// TwinCAT 3 PLC project HARTL_PowerLink_v2_01
// ProgramVersion: 3.1.4023.0
// libraries:
//   EfficientIO Communicator, * (EfficientIO)
//   EfficientIO ModbusTCP, * (EfficientIO)
//   Lynus Energy Basic, * (Lynus AG)
//   Lynus Standards, * (Lynus AG)
//   Tc2_BABasic, * (Beckhoff Automation GmbH)
//   Tc2_ModbusSrv, * (Beckhoff Automation GmbH)
//   Tc2_Standard, * (Beckhoff Automation GmbH)
//   Tc2_System, * (Beckhoff Automation GmbH)
//   Tc2_Utilities, * (Beckhoff Automation GmbH)
//   Tc3_Module, * (Beckhoff Automation GmbH)
// project tree:
//   / FastTask.TcTTO (not stored), MiddleTask.TcTTO, SlowTask.TcTTO
//   FBs/ FB_EM24_DIN.TcPOU, FB_Enphase.TcPOU (not stored), FB_Enphase_Helper.TcPOU, FB_ModBus_2Registers.TcPOU
//   POUs/ prgBattery.TcPOU, prgCalc.TcPOU, prgComEffIO.TcPOU, prgEM.TcPOU, prgEMS.TcPOU, prgEnphase.TcPOU (not stored), prgPV.TcPOU, prgCS.TcPOU, prgRWEffIO.TcPOU (not stored), prgSystemTime.TcPOU, prgVarEffIO.TcPOU (not stored)
// real-time tasks:
//   TASK MiddleTask: cycle T#10ms, priority 20, ADS port 350
//   TASK FastTask: cycle T#5ms, priority 19, ADS port 351
//   TASK SlowTask: cycle T#20ms, priority 21, ADS port 352
// I/O:
//   DEVICE Device 1 (Beckhoff CCAT)
//   DEVICE Device 2 (CX-BK)
//     Box 1 (CX-BK)
// variable links:
//   HARTL_PowerLink_v2_01/HARTL_PowerLink_v2_01 Instance <-> Device 2 (CX-BK)/Box 1 (CX-BK)
//     MiddleTask Inputs/prgEM.fbEM1.fbKL3403.byStateCH1 <-> Term 2 (KL3403)/Channel 1/State
//     MiddleTask Inputs/prgEM.fbEM1.fbKL3403.byStateCH2 <-> Term 2 (KL3403)/Channel 2/State
//     MiddleTask Inputs/prgEM.fbEM1.fbKL3403.byStateCH3 <-> Term 2 (KL3403)/Channel 3/State
//     MiddleTask Inputs/prgEM.fbEM2.fbKL3403.byStateCH1 <-> Term 3 (KL3403)/Channel 1/State
//     MiddleTask Inputs/prgEM.fbEM2.fbKL3403.byStateCH2 <-> Term 3 (KL3403)/Channel 2/State
//     MiddleTask Inputs/prgEM.fbEM2.fbKL3403.byStateCH3 <-> Term 3 (KL3403)/Channel 3/State
//     MiddleTask Inputs/prgEM.fbEM3.fbKL3403.byStateCH1 <-> Term 4 (KL3403)/Channel 1/State
//     MiddleTask Inputs/prgEM.fbEM3.fbKL3403.byStateCH2 <-> Term 4 (KL3403)/Channel 2/State
//     MiddleTask Inputs/prgEM.fbEM3.fbKL3403.byStateCH3 <-> Term 4 (KL3403)/Channel 3/State
//     MiddleTask Inputs/prgEM.fbEM4.fbKL3403.byStateCH1 <-> Term 5 (KL3403)/Channel 1/State
//     MiddleTask Inputs/prgEM.fbEM4.fbKL3403.byStateCH2 <-> Term 5 (KL3403)/Channel 2/State
//     MiddleTask Inputs/prgEM.fbEM4.fbKL3403.byStateCH3 <-> Term 5 (KL3403)/Channel 3/State
//     MiddleTask Inputs/prgEM.fbEM1.fbKL3403.iDataInCH1 <-> Term 2 (KL3403)/Channel 1/Data In
//     MiddleTask Inputs/prgEM.fbEM1.fbKL3403.iDataInCH2 <-> Term 2 (KL3403)/Channel 2/Data In
//     MiddleTask Inputs/prgEM.fbEM1.fbKL3403.iDataInCH3 <-> Term 2 (KL3403)/Channel 3/Data In
//     MiddleTask Inputs/prgEM.fbEM2.fbKL3403.iDataInCH1 <-> Term 3 (KL3403)/Channel 1/Data In
//     MiddleTask Inputs/prgEM.fbEM2.fbKL3403.iDataInCH2 <-> Term 3 (KL3403)/Channel 2/Data In
//     MiddleTask Inputs/prgEM.fbEM2.fbKL3403.iDataInCH3 <-> Term 3 (KL3403)/Channel 3/Data In
//     MiddleTask Inputs/prgEM.fbEM3.fbKL3403.iDataInCH1 <-> Term 4 (KL3403)/Channel 1/Data In
//     MiddleTask Inputs/prgEM.fbEM3.fbKL3403.iDataInCH2 <-> Term 4 (KL3403)/Channel 2/Data In
//     MiddleTask Inputs/prgEM.fbEM3.fbKL3403.iDataInCH3 <-> Term 4 (KL3403)/Channel 3/Data In
//     MiddleTask Inputs/prgEM.fbEM4.fbKL3403.iDataInCH1 <-> Term 5 (KL3403)/Channel 1/Data In
//     MiddleTask Inputs/prgEM.fbEM4.fbKL3403.iDataInCH2 <-> Term 5 (KL3403)/Channel 2/Data In
//     MiddleTask Inputs/prgEM.fbEM4.fbKL3403.iDataInCH3 <-> Term 5 (KL3403)/Channel 3/Data In
//     MiddleTask Inputs/prgEM.fbKBusState.uiKBusState_OUT <-> Inputs/State
//     MiddleTask Outputs/prgEM.fbEM1.fbKL3403.byCntrCH1 <-> Term 2 (KL3403)/Channel 1/Ctrl
//     MiddleTask Outputs/prgEM.fbEM1.fbKL3403.byCntrCH2 <-> Term 2 (KL3403)/Channel 2/Ctrl
//     MiddleTask Outputs/prgEM.fbEM1.fbKL3403.byCntrCH3 <-> Term 2 (KL3403)/Channel 3/Ctrl
//     MiddleTask Outputs/prgEM.fbEM2.fbKL3403.byCntrCH1 <-> Term 3 (KL3403)/Channel 1/Ctrl
//     MiddleTask Outputs/prgEM.fbEM2.fbKL3403.byCntrCH2 <-> Term 3 (KL3403)/Channel 2/Ctrl
//     MiddleTask Outputs/prgEM.fbEM2.fbKL3403.byCntrCH3 <-> Term 3 (KL3403)/Channel 3/Ctrl
//     MiddleTask Outputs/prgEM.fbEM3.fbKL3403.byCntrCH1 <-> Term 4 (KL3403)/Channel 1/Ctrl
//     MiddleTask Outputs/prgEM.fbEM3.fbKL3403.byCntrCH2 <-> Term 4 (KL3403)/Channel 2/Ctrl
//     MiddleTask Outputs/prgEM.fbEM3.fbKL3403.byCntrCH3 <-> Term 4 (KL3403)/Channel 3/Ctrl
//     MiddleTask Outputs/prgEM.fbEM4.fbKL3403.byCntrCH1 <-> Term 5 (KL3403)/Channel 1/Ctrl
//     MiddleTask Outputs/prgEM.fbEM4.fbKL3403.byCntrCH2 <-> Term 5 (KL3403)/Channel 2/Ctrl
//     MiddleTask Outputs/prgEM.fbEM4.fbKL3403.byCntrCH3 <-> Term 5 (KL3403)/Channel 3/Ctrl
//     MiddleTask Outputs/prgEMS.bQ1State <-> Term 6 (KL2012)/Channel 1/Output
//     MiddleTask Outputs/prgEMS.bQ2State <-> Term 6 (KL2012)/Channel 2/Output
//     MiddleTask Outputs/prgEMS.bQ3State <-> Term 7 (KL2012)/Channel 1/Output
//     MiddleTask Outputs/prgEMS.bQ4State <-> Term 7 (KL2012)/Channel 2/Output

CONFIGURATION HARTL_PowerLink_v2_01
    RESOURCE PLC ON TwinCAT3
        TASK MiddleTask(INTERVAL := T#10ms, PRIORITY := 20);
        TASK SlowTask(INTERVAL := T#20ms, PRIORITY := 21);
        PROGRAM prgEM WITH MiddleTask : prgEM;
        PROGRAM prgEMS WITH MiddleTask : prgEMS;
        PROGRAM prgSystemTime WITH MiddleTask : prgSystemTime;
        PROGRAM prgCS WITH MiddleTask : prgCS;
        PROGRAM prgCalc WITH MiddleTask : prgCalc;
        PROGRAM prgComEffIO WITH SlowTask : prgComEffIO;
    END_RESOURCE
END_CONFIGURATION

// ---- POUs/prgEM.TcPOU
PROGRAM prgEM
VAR
	fbKBusState		: FB_K_Bus_State;
	fbEM1			: FB_EM_Beckhoff_KL3403;
	fbEM1Counter	: FB_EnergyCounter;
	fbEM2			: FB_EM_Beckhoff_KL3403;
	fbEM2Counter	: FB_EnergyCounter;
	fbEM3			: FB_EM_Beckhoff_KL3403;
	fbEM3Counter	: FB_EnergyCounter;
	fbEM4			: FB_EM_Beckhoff_KL3403;
	fbEM4Counter	: FB_EnergyCounter;
	lrPowerEM1		: LREAL;						//{#lynus.ag#()}
	lrPowerEM2		: LREAL;						//{#lynus.ag#()}
	lrPowerEM3		: LREAL;						//{#lynus.ag#()}
	lrPowerEM4		: LREAL;						//{#lynus.ag#()}
	lr_InputVoltage_L1N		: LREAL;						//{#lynus.ag#()}
	lr_InputVoltage_L2N		: LREAL;						//{#lynus.ag#()}
	lr_InputVoltage_L3N		: LREAL;						//{#lynus.ag#()}
	lr_InputVoltage_L1L2	: LREAL;						//{#lynus.ag#()}
	lr_InputVoltage_L2L3	: LREAL;						//{#lynus.ag#()}
	lr_InputVoltage_L3L1	: LREAL;						//{#lynus.ag#()}


END_VAR
VAR PERSISTENT
	lrCounterEM1	: LREAL;						//{#lynus.ag#()}
	lrCounterEM2	: LREAL;						//{#lynus.ag#()}
	lrCounterEM3	: LREAL;						//{#lynus.ag#()}
	lrCounterEM4	: LREAL;						//{#lynus.ag#()}
END_VAR

fbKBusState(uiKBusState_OUT=> );

// Base Connection

fbEM1(
	bEnable:= TRUE, 
	bChannel1Invers:= FALSE,
	bChannel2Invers:= FALSE,
	bChannel3Invers:= FALSE,
	uiCurrentTransformerRatioL1:= 64, 
	uiCurrentTransformerRatioL2:= 64, 
	uiCurrentTransformerRatioL3:= 64, 
	uiKBusState_IN:= fbKBusState.uiKBusState_OUT, 
	stDataEMPower=> , 
	stDataEMCounter=> , 
	stDataEMPowerRealTime=> , 
	stDataEMCounterRealTime=> , 
	diNrOfEM_OUT=> );

lrPowerEM1 := fbEM1.stDataEMPower.lrPowerTotal;	
lr_InputVoltage_L1N := fbEM1.stDataEMPower.lrVoltageL1N;
lr_InputVoltage_L2N := fbEM1.stDataEMPower.lrVoltageL2N;
lr_InputVoltage_L3N := fbEM1.stDataEMPower.lrVoltageL3N;
lr_InputVoltage_L1L2 := fbEM1.stDataEMPower.lrVoltageL1L2;
lr_InputVoltage_L2L3 := fbEM1.stDataEMPower.lrVoltageL2L3;
lr_InputVoltage_L3L1 := fbEM1.stDataEMPower.lrVoltageL3L1;

fbEM1Counter(
	byActiveTariff:= 1, 
	lrPowerInput:= lrPowerEM1, 
	lrTotalCounterEnergy_Consumption=> , 
	lrTotalCounterEnergy_Production=> , 
	lrCounterEnergyT1_Consumption=> , 
	lrCounterEnergyT2_Consumption=> , 
	lrCounterEnergyT1_Production=> , 
	lrCounterEnergyT2_Production=> );
	
IF fbEM1Counter.lrTotalCounterEnergy_Consumption > lrCounterEM1 THEN  	
	lrCounterEM1 := fbEM1Counter.lrTotalCounterEnergy_Consumption;
END_IF

// Output1, 3x400V 32A, CEE32

fbEM2(
	bEnable:= TRUE, 
	bChannel1Invers:= FALSE,
	bChannel2Invers:= FALSE,
	bChannel3Invers:= FALSE,
	uiCurrentTransformerRatioL1:= 35, 
	uiCurrentTransformerRatioL2:= 35, 
	uiCurrentTransformerRatioL3:= 35, 
	uiKBusState_IN:= fbKBusState.uiKBusState_OUT, 
	stDataEMPower=> , 
	stDataEMCounter=> , 
	stDataEMPowerRealTime=> , 
	stDataEMCounterRealTime=> , 
	diNrOfEM_OUT=> );

lrPowerEM2 := fbEM2.stDataEMPower.lrPowerTotal;	

fbEM2Counter(
	byActiveTariff:= 1, 
	lrPowerInput:= lrPowerEM2, 
	lrTotalCounterEnergy_Consumption=> , 
	lrTotalCounterEnergy_Production=> , 
	lrCounterEnergyT1_Consumption=> , 
	lrCounterEnergyT2_Consumption=> , 
	lrCounterEnergyT1_Production=> , 
	lrCounterEnergyT2_Production=> );
	
IF fbEM2Counter.lrTotalCounterEnergy_Consumption > lrCounterEM2 THEN  	
	lrCounterEM2 := fbEM2Counter.lrTotalCounterEnergy_Consumption;
END_IF


// Output2, 3x400V 32A, CEE32

fbEM3(
	bEnable:= TRUE, 
	bChannel1Invers:= FALSE,
	bChannel2Invers:= FALSE,
	bChannel3Invers:= FALSE,
	uiCurrentTransformerRatioL1:= 35, 
	uiCurrentTransformerRatioL2:= 35, 
	uiCurrentTransformerRatioL3:= 35, 
	uiKBusState_IN:= fbKBusState.uiKBusState_OUT, 
	stDataEMPower=> , 
	stDataEMCounter=> , 
	stDataEMPowerRealTime=> , 
	stDataEMCounterRealTime=> , 
	diNrOfEM_OUT=> );

lrPowerEM3 := fbEM3.stDataEMPower.lrPowerTotal;	

fbEM3Counter(
	byActiveTariff:= 1, 
	lrPowerInput:= lrPowerEM3, 
	lrTotalCounterEnergy_Consumption=> , 
	lrTotalCounterEnergy_Production=> , 
	lrCounterEnergyT1_Consumption=> , 
	lrCounterEnergyT2_Consumption=> , 
	lrCounterEnergyT1_Production=> , 
	lrCounterEnergyT2_Production=> );
	
IF fbEM3Counter.lrTotalCounterEnergy_Consumption > lrCounterEM3 THEN  	
	lrCounterEM3 := fbEM3Counter.lrTotalCounterEnergy_Consumption;
END_IF


// Output3, 3x400V 16A, CEE16

fbEM4(
	bEnable:= TRUE, 
	bChannel1Invers:= FALSE,
	bChannel2Invers:= FALSE,
	bChannel3Invers:= FALSE,
	uiCurrentTransformerRatioL1:= 35, 
	uiCurrentTransformerRatioL2:= 35, 
	uiCurrentTransformerRatioL3:= 35, 
	uiKBusState_IN:= fbKBusState.uiKBusState_OUT, 
	stDataEMPower=> , 
	stDataEMCounter=> , 
	stDataEMPowerRealTime=> , 
	stDataEMCounterRealTime=> , 
	diNrOfEM_OUT=> );

lrPowerEM4 := fbEM4.stDataEMPower.lrPowerTotal;	

fbEM4Counter(
	byActiveTariff:= 1, 
	lrPowerInput:= lrPowerEM4, 
	lrTotalCounterEnergy_Consumption=> , 
	lrTotalCounterEnergy_Production=> , 
	lrCounterEnergyT1_Consumption=> , 
	lrCounterEnergyT2_Consumption=> , 
	lrCounterEnergyT1_Production=> , 
	lrCounterEnergyT2_Production=> );
	
IF fbEM4Counter.lrTotalCounterEnergy_Consumption > lrCounterEM4 THEN  	
	lrCounterEM4 := fbEM4Counter.lrTotalCounterEnergy_Consumption;
END_IF

END_PROGRAM

// ---- POUs/prgEMS.TcPOU
PROGRAM prgEMS
VAR
	// Q1, 3x400V 32A, CEE32
	fbQ1						: FB_Light;
	bQ1On						: BOOL;						//{#lynus.ag#()}
	bQ1Off						: BOOL;						//{#lynus.ag#()}
	bQ1State	AT%Q*			: BOOL;						//{#lynus.ag#()}
	// Q2, 3x400V 32A, CEE32
	fbQ2						: FB_Light;
	bQ2On						: BOOL;						//{#lynus.ag#()}
	bQ2Off						: BOOL;						//{#lynus.ag#()}
	bQ2State	AT%Q*			: BOOL;						//{#lynus.ag#()}
	// Q3, 3x400V 16A, CEE16
	fbQ3						: FB_Light;	
	bQ3On						: BOOL;						//{#lynus.ag#()}
	bQ3Off						: BOOL;						//{#lynus.ag#()}
	bQ3State	AT%Q*			: BOOL;						//{#lynus.ag#()}
	// Q4, 3x400V 16A, CEE16, EV Charging
	fbQ4						: FB_Light;
	bQ4On						: BOOL;						//{#lynus.ag#()}
	bQ4Off						: BOOL;						//{#lynus.ag#()}
	bQ4State	AT%Q*			: BOOL;						//{#lynus.ag#()}
	
	// Automatic PV-Inverter Shutdown
	fbNFS_PV					: FB_WeeklyTimeSwitch;
	fbCalcSunriseSunset   		: FB_CalcSunriseSunset;
	todSunrise            		: TOD;
	todSunset             		: TOD;
END_VAR
VAR PERSISTENT
	bEnableNFS_PV				: BOOL;						//{#lynus.ag#()}
END_VAR

// To-Do:
// adopt Longitude and Latitude
// set bEdgeOn and bEdgeOff to correct Q Variables


// Output Controls
fbQ1(bOn:=bQ1On, bOff:=bQ1Off, bLight=>bQ1State);
fbQ2(bOn:=bQ2On, bOff:=bQ2Off, bLight=>bQ2State);
fbQ3(bOn:=bQ3On, bOff:=bQ3Off, bLight=>bQ3State);
fbQ4(bOn:=bQ4On, bOff:=bQ4Off, bLight=>bQ4State);

// Sunrise, Sunset calc
IF prgSystemTime.bSystemTimeValid THEN

	fbCalcSunriseSunset(
		fDegreeOfLongitude := 11.5820,   (* Longitude of Munich, Lochhausen *)
        fDegreeOfLatitude := 48.1351,   (* Latitude of Munich, Lochhausen *)
    	fReferenceMeridian := 15.0,  (* Central European Time *)
        dCurrentDate := DT_TO_DATE(prgSystemTime.dtSystemTime),
        todSunrise => todSunrise,
        todSunset => todSunset);
END_IF

// Automatic PV-Inverter Shutdown
IF prgSystemTime.bSystemTimeValid THEN
	fbNFS_PV(
		bEnable:=bEnableNFS_PV, 
		tCurrentDateTime:=prgSystemTime.dtSystemTime, 
		tSwitchOnTime:=todSunrise, 
		tSwitchOffTime:=todSunset, 
		bSunday:=TRUE, 
		bMonday:=TRUE, 
		bTuesday:=TRUE, 
		bWednesday:=TRUE, 
		bThursday:=TRUE, 
		bFriday:=TRUE, 
		bSaturday:=TRUE,
		bEdgeOn=> ,
		bEdgeOff=> );
END_IF

END_PROGRAM

// ---- POUs/prgSystemTime.TcPOU
PROGRAM prgSystemTime
VAR
	fbGetTime			: NT_GetTime;
	dtSystemTime		: DT;
	stDateTime			: TIMESTRUCT;
	tonGetTime			: TON;
	nStep				: INT;
	bSystemTimeValid	: BOOL := FALSE;
END_VAR

CASE nStep OF
0:
	tonGetTime(IN:=TRUE, PT:=T#500MS);
	IF (tonGetTime.Q) THEN
		tonGetTime(IN := FALSE);
		nStep:=10;
	END_IF

10:
	fbGetTime(NETID:='', START:=TRUE, TMOUT:=T#2S);
	IF (NOT fbGetTime.BUSY) THEN
		stDateTime := fbGetTime.TIMESTR;
		dtSystemTime := SYSTEMtimE_TO_DT(fbGetTime.TIMESTR);
		fbGetTime(START := FALSE);
		bSystemTimeValid := TRUE;
		nStep := 0;
	END_IF	
END_CASE

END_PROGRAM

// ---- POUs/prgCS.TcPOU
PROGRAM prgCS
VAR
	fbCS						: FB_EM24_DIN;
	fbCSCounter					: FB_EnergyCounter;
	lrPowerCS					: LREAL;						//{#lynus.ag#()}
	// udintErrorWarningCS			: UDINT;
END_VAR
VAR PERSISTENT
	lrCounterCS					: LREAL;						//{#lynus.ag#()}
	lrCounterCSeIO				: LREAL;						//{#lynus.ag#()}
END_VAR

// To-Do:
// adopt FB Declaration, change to new FB for ENERGYMID
// adopt FB Definition, change to correct in/out Vars for ENERGYMID
// correct lrPowerCS definition
// correct lrCounterCS definition
// correct byErrorWarningCS definition

fbCS(
	m_Enable:= TRUE, 
	str_IPAdress:= '192.168.1.20',  
	real_RealPower_kW=> lrPowerCS, 
	real_RealPowerL1_kW=> , 
	real_RealPowerL2_kW=> , 
	real_RealPowerL3_kW=> , 
	real_ReactivePower_kVAr=> , 
	real_ApparentPower_kVA=> , 
	real_Frequency_Hz=> , 
	real_VoltageL1N_V=> , 
	real_VoltageL2N_V=> , 
	real_VoltageL3N_V=> , 
	real_VoltageL1L2_V=> , 
	real_VoltageL2L3_V=> , 
	real_VoltageL3L1_V=> , 
	real_CurrentL1_A=> , 
	real_CurrentL2_A=> , 
	real_CurrentL3_A=> , 
	real_EnergyTotal_Import_kWh=> , 
	real_EnergyTotal_Export_kWh=> , 
	real_EnergyTotal_ExportT1_kWh=> , 
	real_EnergyTotal_ExportT2_kWh=> , 
	real_EnergyTotal_ExportT3_kWh=> , 
	real_EnergyTotal_ExportT4_kWh=> , 
	m_PollSuccessful=> , 
	udint_Error_ID=> );



// uErrorWarningCS := fbCS.udint_Error_ID;

// MID conform Counter, read from Energymeter
IF fbCS.real_EnergyTotal_Import_kWh > lrCounterCS THEN  	
	lrCounterCS := fbCS.real_EnergyTotal_Import_kWh;
END_IF

// internal Counter, for comparing purpose
fbCSCounter(
	byActiveTariff:= 1, 
	lrPowerInput:= lrPowerCS, 
	lrTotalCounterEnergy_Consumption=> , 
	lrTotalCounterEnergy_Production=> , 
	lrCounterEnergyT1_Consumption=> , 
	lrCounterEnergyT2_Consumption=> , 
	lrCounterEnergyT1_Production=> , 
	lrCounterEnergyT2_Production=> );
	
IF fbCSCounter.lrTotalCounterEnergy_Consumption > lrCounterCSeIO THEN  	
	lrCounterCSeIO := fbCSCounter.lrTotalCounterEnergy_Consumption;
END_IF

END_PROGRAM

// ---- FBs/FB_EM24_DIN.TcPOU
FUNCTION_BLOCK FB_EM24_DIN
VAR_INPUT PERSISTENT
	m_Enable					: BOOL;						//Enable the Fuctionblock and his logic
	str_IPAdress				: STRING(15);				//IP Adress of the meter
END_VAR
VAR_OUTPUT
	real_RealPower_kW				: REAL;					// Real power in W
	real_RealPowerL1_kW				: REAL;					// Real power in W
	real_RealPowerL2_kW				: REAL;					// Real power in W
	real_RealPowerL3_kW				: REAL;					// Real power in W
	real_ReactivePower_kVAr			: REAL;					// Reactive power in VAr
	real_ApparentPower_kVA			: REAL;					// Apparent power in VA
	real_Frequency_Hz				: REAL;					// Frequency in Hz
	real_VoltageL1N_V				: REAL;					//  Voltage L1-N in V 
	real_VoltageL2N_V				: REAL;					//  Voltage L2-N in V 
	real_VoltageL3N_V				: REAL;					//  Voltage L3-N in V 
	real_VoltageL1L2_V				: REAL;					//  Voltage L1-L2 in V 
	real_VoltageL2L3_V				: REAL;					//  Voltage L2-L3 in V 
	real_VoltageL3L1_V				: REAL;					//  Voltage L3-L1 in V 
	real_CurrentL1_A				: REAL;					//  Current L1 in A
	real_CurrentL2_A				: REAL;					//  Current L2 in A
	real_CurrentL3_A				: REAL;					//  Current L3 in A
	real_EnergyTotal_Import_kWh		: REAL;					// Energy total in Wh
	real_EnergyTotal_Export_kWh		: REAL;					// Energy total in Wh
	real_EnergyTotal_ExportT1_kWh	: REAL;					// Energy total in Wh
	real_EnergyTotal_ExportT2_kWh	: REAL;					// Energy total in Wh
	real_EnergyTotal_ExportT3_kWh	: REAL;					// Energy total in Wh
	real_EnergyTotal_ExportT4_kWh	: REAL;					// Energy total in Wh
	
	m_PollSuccessful				: BOOL;					// Poll succesfull		
	udint_Error_ID					: UDINT;				// ERR ID FB_MBReadRegs
END_VAR
VAR
	{attribute 'hide'}
	w_Adress					: WORD;						//modbus adress
	{attribute 'hide'}
	usint_Quantity				: USINT;					//Number of Words to get polled, max 100
	{attribute 'hide'}
	fbConvertWordToDword		: FB_CV_WORD_TO_DWORD;			//Convert Word to Dword
	{attribute 'hide'}
	usintSign					: USINT;						// converstion dword to real	
	{attribute 'hide'}
	intExponent					: INT;							// converstion dword to real
	{attribute 'hide'}
	realMantisse				: REAL;							// converstion dword to real
	{attribute 'hide'}
	timer_Delay					: TON;						//Timer for Delay between Requests
	{attribute 'hide'}
	timer_DelayStart			: TON;						//Timer to start the state machine with Delay after enabling or after the system ist restartet
	{attribute 'hide'}
	timer_TimeOut				: TON;						//Timer for Timeout MB Read
	{attribute 'hide'}
	iStateModbusRead			: INT;						//State machine for read out Data over Modbus RTU
	{attribute 'hide'}
	fbMBRead_FC3				: FB_MBReadRegs  ;		//Modbus Read Function (FC3)
	{attribute 'hide'}
	ftrig_PEnable				: f_trig;					//Internal positive Edge
	{attribute 'hide'}
	iStateModbusError			: INT;						//State machine for error out Data over Modbus TCP/IP	
	{attribute 'hide'}
	FPError_FC_3				: R_TRIG;					//Internal positive Edge
	{attribute 'hide'}
	arrBuffer_FC3				: ARRAY[0..10] OF WORD;		//Buffer with Data from FC3
	{attribute 'hide'}
	arrBuffer_Received			: ARRAY[0..120] OF WORD;		//Total received Data
	{attribute 'hide'}
	timer_Connection_ok			: TON;
	{attribute 'hide'}
	int_Data_Received			: INT;
	{attribute 'hide'}
	m_MBTCPError				: BOOL;
	{attribute 'hide'}
	int_Data_Received_old		: INT;
	{attribute 'hide'}
	timer_Connection_ok_TOF	: TOF;
	{attribute 'hide'}
	m_Poll_ok: BOOL;
	{attribute 'hide'}
	timer_Wait: Ton;
	{attribute 'hide'}
	int_TimeoutError: INT;
	{attribute 'hide'}
	int_FC4Error: INT;
	{attribute 'hide'}
	i: INT;
END_VAR

// v0.1 by Stefan Lackner 20230330
// tested, but not with current flowing. Votlages & frequency working.
// reads out Carlo Gavazzi EM24-Din Multimeter


(*--------------------------------------------------------------------------------------------Limits-------------------------------------------------------------------------------------*)
w_Adress := LIMIT(0,w_Adress,65000);
usint_Quantity := LIMIT(1,usint_Quantity,100);
	
(*--------------------------------------------------------------------------------------------State Machine Read--------------------------------------------------------------------------------------*)

//Timer for Delay
timer_Delay(IN:= , PT:= T#50MS, Q=> , ET=> );

//Timeout Timer is dissabled when the Init Step is aktiv or the function is not enabled
IF iStateModbusRead = 0 OR NOT m_Enable THEN 
	timer_Timeout.IN := FALSE; 
END_IF
timer_Timeout(IN:= , PT:= T#1S, Q=> , ET=> );

//Enable with Delay that not all sockets have to be created at the same time
timer_DelayStart(IN:= m_Enable, PT:= T#1S, Q=> , ET=> );
ftrig_PEnable(CLK:= timer_DelayStart.Q, Q=> );

IF ftrig_PEnable.Q AND iStateModbusRead = 0 THEN 
	iStateModbusRead := 1; 
END_IF		
		
//Not Enabled
IF NOT m_Enable THEN 
	iStateModbusRead := 0; 
	iStateModbusError := 0; 
END_IF		
		
CASE iStateModbusRead OF

	0://Init Step 
		timer_Delay.IN := FALSE;
		fbMBRead_FC3.bExecute := FALSE;
		m_Poll_ok:=FALSE;
		int_Data_Received:=0;
		iStateModbusRead := iStateModbusRead+1;

	1: // clean the array  Poll 1
		FOR i:=0 TO 10 BY 1 DO
			arrBuffer_FC3[i] := 0;
		END_FOR
		w_Adress := 0;
		usint_Quantity := 10; 
		iStateModbusRead := iStateModbusRead+1;
		
	2://read the required registers
		//Start Read Poll 1
		fbMBRead_FC3.nQuantity := usint_Quantity;
		fbMBRead_FC3.nMBAddr := w_Adress;
		fbMBRead_FC3.bExecute := TRUE;
		fbMBRead_FC3.nUnitID := 1;
		timer_Timeout.IN := TRUE;
		IF fbMBRead_FC3.bBusy THEN 
			timer_Delay.IN := TRUE; 
		END_IF
		
		//Wait for Delay, copy Data and then next step
		IF NOT fbMBRead_FC3.bBusy AND NOT fbMBRead_FC3.bError AND timer_Delay.Q THEN
			m_Poll_ok:=TRUE;
			int_Data_Received:=int_Data_Received+1;
			m_MBTCPError := FALSE; 
			
			FOR i:=0 TO 9 BY 1 DO
				arrBuffer_Received[i + WORD_TO_INT(w_Adress)] := arrBuffer_FC3[i];
			END_FOR
			
			//Go to Next Step
			timer_Timeout.IN := FALSE;
			fbMBRead_FC3.bExecute := FALSE;
			timer_Delay.IN := FALSE;		
			iStateModbusRead := iStateModbusRead+1;
		END_IF	

		//Error or Timeout
		IF FPError_FC_3.Q THEN 
			iStateModbusError := 300;
			int_FC4Error := int_FC4Error+1;
		ELSIF timer_Timeout.Q THEN  
			timer_Timeout.IN := FALSE; 	
			iStateModbusError := 300;
			int_TimeoutError := int_TimeoutError+1;
		END_IF
	
	3://Wait and go to next step
		timer_Wait.IN := TRUE;
		
		IF timer_Wait.Q = TRUE THEN
			iStateModbusRead := iStateModbusRead+1;
			timer_Wait.IN :=FALSE;
		END_IF

	4: // clean the array  Poll 2
		FOR i:=0 TO 10 BY 1 DO
			arrBuffer_FC3[i] := 0;
		END_FOR
		w_Adress := w_Adress + 10;;
		usint_Quantity := 10; 
		iStateModbusRead := iStateModbusRead+1;
		
	5://read the required registers
		//Start Read Poll 2
		fbMBRead_FC3.nQuantity := usint_Quantity;
		fbMBRead_FC3.nMBAddr := w_Adress;
		fbMBRead_FC3.bExecute := TRUE;
		fbMBRead_FC3.nUnitID := 1;
		timer_Timeout.IN := TRUE;
		IF fbMBRead_FC3.bBusy THEN 
			timer_Delay.IN := TRUE; 
		END_IF
		
		//Wait for Delay, copy Data and then next step
		IF NOT fbMBRead_FC3.bBusy AND NOT fbMBRead_FC3.bError AND timer_Delay.Q THEN
			m_Poll_ok:=TRUE;
			int_Data_Received:=int_Data_Received+1;
			m_MBTCPError := FALSE; 
			
			FOR i:=0 TO 9 BY 1 DO
				arrBuffer_Received[i + WORD_TO_INT(w_Adress)] := arrBuffer_FC3[i];
			END_FOR
			
			//Go to Next Step
			timer_Timeout.IN := FALSE;
			fbMBRead_FC3.bExecute := FALSE;
			timer_Delay.IN := FALSE;		
			iStateModbusRead := iStateModbusRead+1;
		END_IF	

		//Error or Timeout
		IF FPError_FC_3.Q THEN 
			iStateModbusError := 300;
			int_FC4Error := int_FC4Error+1;
		ELSIF timer_Timeout.Q THEN  
			timer_Timeout.IN := FALSE; 	
			iStateModbusError := 300;
			int_TimeoutError := int_TimeoutError+1;
		END_IF
	
	6://Wait and go to next step
		timer_Wait.IN := TRUE;
		
		IF timer_Wait.Q = TRUE THEN
			iStateModbusRead := iStateModbusRead+1;
			timer_Wait.IN :=FALSE;
		END_IF
		
	7: // clean the array  Poll 3
		FOR i:=0 TO 10 BY 1 DO
			arrBuffer_FC3[i] := 0;
		END_FOR
		w_Adress := w_Adress + 10;
		usint_Quantity := 10; 
		iStateModbusRead := iStateModbusRead+1;
		
	8://read the required registers
		//Start Read Poll 3
		fbMBRead_FC3.nQuantity := usint_Quantity;
		fbMBRead_FC3.nMBAddr := w_Adress;
		fbMBRead_FC3.bExecute := TRUE;
		fbMBRead_FC3.nUnitID := 1;
		timer_Timeout.IN := TRUE;
		IF fbMBRead_FC3.bBusy THEN 
			timer_Delay.IN := TRUE; 
		END_IF
		
		//Wait for Delay, copy Data and then next step
		IF NOT fbMBRead_FC3.bBusy AND NOT fbMBRead_FC3.bError AND timer_Delay.Q THEN
			m_Poll_ok:=TRUE;
			int_Data_Received:=int_Data_Received+1;
			m_MBTCPError := FALSE; 
			
			FOR i:=0 TO 9 BY 1 DO
				arrBuffer_Received[i + WORD_TO_INT(w_Adress)] := arrBuffer_FC3[i];
			END_FOR
			
			//Go to Next Step
			timer_Timeout.IN := FALSE;
			fbMBRead_FC3.bExecute := FALSE;
			timer_Delay.IN := FALSE;		
			iStateModbusRead := iStateModbusRead+1;
		END_IF	

		//Error or Timeout
		IF FPError_FC_3.Q THEN 
			iStateModbusError := 300;
			int_FC4Error := int_FC4Error+1;
		ELSIF timer_Timeout.Q THEN  
			timer_Timeout.IN := FALSE; 	
			iStateModbusError := 300;
			int_TimeoutError := int_TimeoutError+1;
		END_IF
	
	9://Wait and go to next step
		timer_Wait.IN := TRUE;
		
		IF timer_Wait.Q = TRUE THEN
			iStateModbusRead := iStateModbusRead+1;
			timer_Wait.IN :=FALSE;
		END_IF
		
	10: // clean the array  Poll 4
		FOR i:=0 TO 10 BY 1 DO
			arrBuffer_FC3[i] := 0;
		END_FOR
		w_Adress := w_Adress + 10;
		usint_Quantity := 10; 
		iStateModbusRead := iStateModbusRead+1;
		
	11://read the required registers
		//Start Read Poll 4
		fbMBRead_FC3.nQuantity := usint_Quantity;
		fbMBRead_FC3.nMBAddr := w_Adress;
		fbMBRead_FC3.bExecute := TRUE;
		fbMBRead_FC3.nUnitID := 1;
		timer_Timeout.IN := TRUE;
		IF fbMBRead_FC3.bBusy THEN 
			timer_Delay.IN := TRUE; 
		END_IF
		
		//Wait for Delay, copy Data and then next step
		IF NOT fbMBRead_FC3.bBusy AND NOT fbMBRead_FC3.bError AND timer_Delay.Q THEN
			m_Poll_ok:=TRUE;
			int_Data_Received:=int_Data_Received+1;
			m_MBTCPError := FALSE; 
			
			FOR i:=0 TO 9 BY 1 DO
				arrBuffer_Received[i + WORD_TO_INT(w_Adress)] := arrBuffer_FC3[i];
			END_FOR
			
			//Go to Next Step
			timer_Timeout.IN := FALSE;
			fbMBRead_FC3.bExecute := FALSE;
			timer_Delay.IN := FALSE;		
			iStateModbusRead := iStateModbusRead+1;
		END_IF	

		//Error or Timeout
		IF FPError_FC_3.Q THEN 
			iStateModbusError := 300;
			int_FC4Error := int_FC4Error+1;
		ELSIF timer_Timeout.Q THEN  
			timer_Timeout.IN := FALSE; 	
			iStateModbusError := 300;
			int_TimeoutError := int_TimeoutError+1;
		END_IF
	
	12://Wait and go to next step
		timer_Wait.IN := TRUE;
		
		IF timer_Wait.Q = TRUE THEN
			iStateModbusRead := iStateModbusRead+1;
			timer_Wait.IN :=FALSE;
		END_IF		
		
	13: // clean the array  Poll 4
		FOR i:=0 TO 10 BY 1 DO
			arrBuffer_FC3[i] := 0;
		END_FOR
		w_Adress := w_Adress + 10;
		usint_Quantity := 10; 
		iStateModbusRead := iStateModbusRead+1;
		
	14://read the required registers
		//Start Read Poll 4
		fbMBRead_FC3.nQuantity := usint_Quantity;
		fbMBRead_FC3.nMBAddr := w_Adress;
		fbMBRead_FC3.bExecute := TRUE;
		fbMBRead_FC3.nUnitID := 1;
		timer_Timeout.IN := TRUE;
		IF fbMBRead_FC3.bBusy THEN 
			timer_Delay.IN := TRUE; 
		END_IF
		
		//Wait for Delay, copy Data and then next step
		IF NOT fbMBRead_FC3.bBusy AND NOT fbMBRead_FC3.bError AND timer_Delay.Q THEN
			m_Poll_ok:=TRUE;
			int_Data_Received:=int_Data_Received+1;
			m_MBTCPError := FALSE; 
			
			FOR i:=0 TO 9 BY 1 DO
				arrBuffer_Received[i + WORD_TO_INT(w_Adress)] := arrBuffer_FC3[i];
			END_FOR
			
			//Go to Next Step
			timer_Timeout.IN := FALSE;
			fbMBRead_FC3.bExecute := FALSE;
			timer_Delay.IN := FALSE;		
			iStateModbusRead := iStateModbusRead+1;
		END_IF	

		//Error or Timeout
		IF FPError_FC_3.Q THEN 
			iStateModbusError := 300;
			int_FC4Error := int_FC4Error+1;
		ELSIF timer_Timeout.Q THEN  
			timer_Timeout.IN := FALSE; 	
			iStateModbusError := 300;
			int_TimeoutError := int_TimeoutError+1;
		END_IF
	
	15://Wait and go to next step
		timer_Wait.IN := TRUE;
		
		IF timer_Wait.Q = TRUE THEN
			iStateModbusRead := iStateModbusRead+1;
			timer_Wait.IN :=FALSE;
		END_IF
		
	16: // clean the array  Poll 5
		FOR i:=0 TO 10 BY 1 DO
			arrBuffer_FC3[i] := 0;
		END_FOR
		w_Adress := w_Adress + 10;
		usint_Quantity := 10; 
		iStateModbusRead := iStateModbusRead+1;
		
	17://read the required registers
		//Start Read Poll 5
		fbMBRead_FC3.nQuantity := usint_Quantity;
		fbMBRead_FC3.nMBAddr := w_Adress;
		fbMBRead_FC3.bExecute := TRUE;
		fbMBRead_FC3.nUnitID := 1;
		timer_Timeout.IN := TRUE;
		IF fbMBRead_FC3.bBusy THEN 
			timer_Delay.IN := TRUE; 
		END_IF
		
		//Wait for Delay, copy Data and then next step
		IF NOT fbMBRead_FC3.bBusy AND NOT fbMBRead_FC3.bError AND timer_Delay.Q THEN
			m_Poll_ok:=TRUE;
			int_Data_Received:=int_Data_Received+1;
			m_MBTCPError := FALSE; 
			
			FOR i:=0 TO 9 BY 1 DO
				arrBuffer_Received[i + WORD_TO_INT(w_Adress)] := arrBuffer_FC3[i];
			END_FOR
			
			//Go to Next Step
			timer_Timeout.IN := FALSE;
			fbMBRead_FC3.bExecute := FALSE;
			timer_Delay.IN := FALSE;		
			iStateModbusRead := iStateModbusRead+1;
		END_IF	

		//Error or Timeout
		IF FPError_FC_3.Q THEN 
			iStateModbusError := 300;
			int_FC4Error := int_FC4Error+1;
		ELSIF timer_Timeout.Q THEN  
			timer_Timeout.IN := FALSE; 	
			iStateModbusError := 300;
			int_TimeoutError := int_TimeoutError+1;
		END_IF
	
	18://Wait and go to next step
		timer_Wait.IN := TRUE;
		
		IF timer_Wait.Q = TRUE THEN
			iStateModbusRead := iStateModbusRead+1;
			timer_Wait.IN :=FALSE;
		END_IF	

	19: // clean the array  Poll 6
		FOR i:=0 TO 10 BY 1 DO
			arrBuffer_FC3[i] := 0;
		END_FOR
		w_Adress := w_Adress + 10;
		usint_Quantity := 10; 
		iStateModbusRead := iStateModbusRead+1;
		
	20://read the required registers
		//Start Read Poll 6
		fbMBRead_FC3.nQuantity := usint_Quantity;
		fbMBRead_FC3.nMBAddr := w_Adress;
		fbMBRead_FC3.bExecute := TRUE;
		fbMBRead_FC3.nUnitID := 1;
		timer_Timeout.IN := TRUE;
		IF fbMBRead_FC3.bBusy THEN 
			timer_Delay.IN := TRUE; 
		END_IF
		
		//Wait for Delay, copy Data and then next step
		IF NOT fbMBRead_FC3.bBusy AND NOT fbMBRead_FC3.bError AND timer_Delay.Q THEN
			m_Poll_ok:=TRUE;
			int_Data_Received:=int_Data_Received+1;
			m_MBTCPError := FALSE; 
			
			FOR i:=0 TO 9 BY 1 DO
				arrBuffer_Received[i + WORD_TO_INT(w_Adress)] := arrBuffer_FC3[i];
			END_FOR
			
			//Go to Next Step
			timer_Timeout.IN := FALSE;
			fbMBRead_FC3.bExecute := FALSE;
			timer_Delay.IN := FALSE;		
			iStateModbusRead := iStateModbusRead+1;
		END_IF	

		//Error or Timeout
		IF FPError_FC_3.Q THEN 
			iStateModbusError := 300;
			int_FC4Error := int_FC4Error+1;
		ELSIF timer_Timeout.Q THEN  
			timer_Timeout.IN := FALSE; 	
			iStateModbusError := 300;
			int_TimeoutError := int_TimeoutError+1;
		END_IF
	
	21://Wait and go to next step
		timer_Wait.IN := TRUE;
		
		IF timer_Wait.Q = TRUE THEN
			iStateModbusRead := iStateModbusRead+1;
			timer_Wait.IN :=FALSE;
		END_IF	
		
	22: // clean the array  Poll 7
		FOR i:=0 TO 10 BY 1 DO
			arrBuffer_FC3[i] := 0;
		END_FOR
		w_Adress := w_Adress + 10;
		usint_Quantity := 10; 
		iStateModbusRead := iStateModbusRead+1;
		
	23://read the required registers
		//Start Read Poll 7
		fbMBRead_FC3.nQuantity := usint_Quantity;
		fbMBRead_FC3.nMBAddr := w_Adress;
		fbMBRead_FC3.bExecute := TRUE;
		fbMBRead_FC3.nUnitID := 1;
		timer_Timeout.IN := TRUE;
		IF fbMBRead_FC3.bBusy THEN 
			timer_Delay.IN := TRUE; 
		END_IF
		
		//Wait for Delay, copy Data and then next step
		IF NOT fbMBRead_FC3.bBusy AND NOT fbMBRead_FC3.bError AND timer_Delay.Q THEN
			m_Poll_ok:=TRUE;
			int_Data_Received:=int_Data_Received+1;
			m_MBTCPError := FALSE; 
			
			FOR i:=0 TO 9 BY 1 DO
				arrBuffer_Received[i + WORD_TO_INT(w_Adress)] := arrBuffer_FC3[i];
			END_FOR
			
			//Go to Next Step
			timer_Timeout.IN := FALSE;
			fbMBRead_FC3.bExecute := FALSE;
			timer_Delay.IN := FALSE;		
			iStateModbusRead := iStateModbusRead+1;
		END_IF	

		//Error or Timeout
		IF FPError_FC_3.Q THEN 
			iStateModbusError := 300;
			int_FC4Error := int_FC4Error+1;
		ELSIF timer_Timeout.Q THEN  
			timer_Timeout.IN := FALSE; 	
			iStateModbusError := 300;
			int_TimeoutError := int_TimeoutError+1;
		END_IF
	
	24://Wait and go to next step
		timer_Wait.IN := TRUE;
		
		IF timer_Wait.Q = TRUE THEN
			iStateModbusRead := iStateModbusRead+1;
			timer_Wait.IN :=FALSE;
		END_IF	

	25: // clean the array  Poll 8
		FOR i:=0 TO 10 BY 1 DO
			arrBuffer_FC3[i] := 0;
		END_FOR
		w_Adress := w_Adress + 10;
		usint_Quantity := 2;		// only 2 possible, otherwise out of the range 
		iStateModbusRead := iStateModbusRead+1;
		
	26://read the required registers
		//Start Read Poll 8
		fbMBRead_FC3.nQuantity := usint_Quantity;
		fbMBRead_FC3.nMBAddr := w_Adress;
		fbMBRead_FC3.bExecute := TRUE;
		fbMBRead_FC3.nUnitID := 1;
		timer_Timeout.IN := TRUE;
		IF fbMBRead_FC3.bBusy THEN 
			timer_Delay.IN := TRUE; 
		END_IF
		
		//Wait for Delay, copy Data and then next step
		IF NOT fbMBRead_FC3.bBusy AND NOT fbMBRead_FC3.bError AND timer_Delay.Q THEN
			m_Poll_ok:=TRUE;
			int_Data_Received:=int_Data_Received+1;
			m_MBTCPError := FALSE; 
			
			FOR i:=0 TO 9 BY 1 DO
				arrBuffer_Received[i + WORD_TO_INT(w_Adress)] := arrBuffer_FC3[i];
			END_FOR
			
			//Go to Next Step
			timer_Timeout.IN := FALSE;
			fbMBRead_FC3.bExecute := FALSE;
			timer_Delay.IN := FALSE;		
			iStateModbusRead := 30;  // convert data
		END_IF	

		//Error or Timeout
		IF FPError_FC_3.Q THEN 
			iStateModbusError := 300;
			int_FC4Error := int_FC4Error+1;
		ELSIF timer_Timeout.Q THEN  
			timer_Timeout.IN := FALSE; 	
			iStateModbusError := 300;
			int_TimeoutError := int_TimeoutError+1;
		END_IF
	

	
	30: // convert data
		real_VoltageL1N_V 	:= WORD_TO_REAL(arrBuffer_Received[0]) /10;
		real_VoltageL2N_V 	:= WORD_TO_REAL(arrBuffer_Received[2]) /10;
		real_VoltageL3N_V 	:= WORD_TO_REAL(arrBuffer_Received[4]) /10;
		real_VoltageL1L2_V 	:= WORD_TO_REAL(arrBuffer_Received[6]) /10;
		real_VoltageL2L3_V 	:= WORD_TO_REAL(arrBuffer_Received[8]) /10;
		real_VoltageL3L1_V 	:= WORD_TO_REAL(arrBuffer_Received[10]) /10;
		
		real_CurrentL1_A	:= (WORD_TO_REAL(arrBuffer_Received[13]) * 65536 + WORD_TO_REAL(arrBuffer_Received[12])) /1000;
		real_CurrentL2_A	:= (WORD_TO_REAL(arrBuffer_Received[15]) * 65536 + WORD_TO_REAL(arrBuffer_Received[14])) /1000;
		real_CurrentL3_A	:= (WORD_TO_REAL(arrBuffer_Received[17]) * 65536 + WORD_TO_REAL(arrBuffer_Received[16])) /1000;
		
		real_RealPowerL1_kW	:= (WORD_TO_REAL(arrBuffer_Received[19]) * 65536 + WORD_TO_REAL(arrBuffer_Received[18])) /10;	
		real_RealPowerL2_kW	:= (WORD_TO_REAL(arrBuffer_Received[21]) * 65536 + WORD_TO_REAL(arrBuffer_Received[20])) /10;	
		real_RealPowerL3_kW	:= (WORD_TO_REAL(arrBuffer_Received[23]) * 65536 + WORD_TO_REAL(arrBuffer_Received[22])) /10;	
		real_RealPower_kW	:= (WORD_TO_REAL(arrBuffer_Received[41]) * 65536 + WORD_TO_REAL(arrBuffer_Received[40])) /10;	
		real_ApparentPower_kVA	:= (WORD_TO_REAL(arrBuffer_Received[43]) * 65536 + WORD_TO_REAL(arrBuffer_Received[42])) /10;	
		real_ReactivePower_kVAr	:= (WORD_TO_REAL(arrBuffer_Received[45]) * 65536 + WORD_TO_REAL(arrBuffer_Received[44])) /10;	

		real_Frequency_Hz	:= WORD_TO_REAL(arrBuffer_Received[51]) /10;
		
		real_EnergyTotal_Import_kWh 	:= (WORD_TO_REAL(arrBuffer_Received[53]) * 65536 + WORD_TO_REAL(arrBuffer_Received[52])) /10;
		real_EnergyTotal_Export_kWh 	:= (WORD_TO_REAL(arrBuffer_Received[79]) * 65536 + WORD_TO_REAL(arrBuffer_Received[78])) /10;
		real_EnergyTotal_ExportT1_kWh 	:= (WORD_TO_REAL(arrBuffer_Received[71]) * 65536 + WORD_TO_REAL(arrBuffer_Received[70])) /10;
		real_EnergyTotal_ExportT2_kWh 	:= (WORD_TO_REAL(arrBuffer_Received[73]) * 65536 + WORD_TO_REAL(arrBuffer_Received[72])) /10;
		real_EnergyTotal_ExportT3_kWh 	:= (WORD_TO_REAL(arrBuffer_Received[75]) * 65536 + WORD_TO_REAL(arrBuffer_Received[74])) /10;
		real_EnergyTotal_ExportT4_kWh 	:= (WORD_TO_REAL(arrBuffer_Received[77]) * 65536 + WORD_TO_REAL(arrBuffer_Received[76])) /10;
		

		// go to next state
		iStateModbusRead := iStateModbusRead+1;		
		
	31://Wait and go to start
		timer_Wait.IN := TRUE;
		
		IF timer_Wait.Q = TRUE THEN
			iStateModbusRead := 1;
			timer_Wait.IN :=FALSE;
		END_IF	

END_CASE

(* wait timer*)

timer_Wait(PT:=T#1S);


(*------------------------------------------------------------------Error and Warning----------------------------------------------------------------------------*)	
 
timer_Connection_ok			(In:=int_Data_Received<>int_Data_Received_old,PT:=T#10S);
timer_Connection_ok_TOF		(In:=NOT(int_Data_Received<>int_Data_Received_old) AND int_Data_Received>3 ,PT:=T#20S);
int_Data_Received_old:=int_Data_Received;
m_PollSuccessful:=NOT timer_Connection_ok.Q AND timer_Connection_ok_TOF.Q ;

(*------------------------------------------------------------------------------------------Modbus TCP Functions---------------------------------------------------------------------------------------------*)

fbMBRead_FC3(	sIPAddr:= str_IPAdress, 
				nTCPPort:= 502,
				cbLength:= SIZEOF(arrBuffer_FC3), 
				pDestAddr:= ADR(arrBuffer_FC3), 
				tTimeout:= T#10S,
				nErrId => udint_Error_ID);

FPError_FC_3(CLK:= fbMBRead_FC3.bError, Q=> );		

(*------------------------------------------------------------------------------------------State Machine Error---------------------------------------------------------------------------------------------*)	

CASE iStateModbusError OF
	
	300://Error
		timer_Wait.IN :=TRUE;
		timer_Delay.IN := FALSE;
		fbMBRead_FC3.bExecute := FALSE;
		m_MBTCPError := TRUE; 		
		m_Poll_ok:=FALSE;
		int_Data_Received:=0;
		
				//Restart from new with the Read out part after an Error
		IF timer_Wait.Q = TRUE THEN
			iStateModbusRead := 0;	
			iStateModbusError := 0;
			timer_Wait.IN :=FALSE;
			timer_Timeout.IN := FALSE;
		END_IF		
							
END_CASE

END_FUNCTION_BLOCK

// ---- POUs/prgCalc.TcPOU
PROGRAM prgCalc
VAR
	fbQ56Counter	: FB_EnergyCounter;
	lrPowerQ56		: LREAL;						//{#lynus.ag#()}
END_VAR
VAR PERSISTENT
	lrCounterQ56	: LREAL;						//{#lynus.ag#()}
	lrCO2Enphase	: LREAL;						//{#lynus.ag#()}
	lrCO2PV			: LREAL;						//{#lynus.ag#()}
END_VAR

// calc Output 5 & 6, 230V 16A, Schuko
// choose one of the two calc-options

// 1 -- if prgPV is in use
// lrPowerQ56 := (prgEM.lrPowerEM1 + prgBattery.lrPowerBatt + prgPV.lrPowerPV) - (prgEM.lrPowerEM2 + prgEM.lrPowerEM3 + prgEM.lrPowerEM4 + prgCS.lrPowerCS);
lrPowerQ56 := (prgEM.lrPowerEM1) - (prgEM.lrPowerEM2 + prgEM.lrPowerEM3 + prgEM.lrPowerEM4 + prgCS.lrPowerCS);

// 2 -- if prgEnphase is in use
// lrPowerQ56 := (prgEM.lrPowerEM1 + prgBattery.lrPowerBatt + prgEnphase.lrPowerPV) - (prgEM.lrPowerEM2 + prgEM.lrPowerEM3 + prgEM.lrPowerEM4 + prgCS.lrPowerCS);

fbQ56Counter(
	byActiveTariff:= 1, 
	lrPowerInput:= lrPowerQ56, 
	lrTotalCounterEnergy_Consumption=> , 
	lrTotalCounterEnergy_Production=> , 
	lrCounterEnergyT1_Consumption=> , 
	lrCounterEnergyT2_Consumption=> , 
	lrCounterEnergyT1_Production=> , 
	lrCounterEnergyT2_Production=> );
	
IF fbQ56Counter.lrTotalCounterEnergy_Consumption > lrCounterQ56 THEN  	
	lrCounterQ56 := fbQ56Counter.lrTotalCounterEnergy_Consumption;
END_IF

// calc saved CO2
// lrCO2Enphase := prgEnphase.lrCounterPV * 0.428;
// lrCO2PV := prgPV.lrCounterPV * 0.428;

END_PROGRAM

// ---- POUs/prgComEffIO.TcPOU
PROGRAM prgComEffIO
VAR
	fbCom		: FB_MqttCommunicator_V2;
END_VAR

fbCom(
	bConnect:= TRUE, 
	strAuthkey := 'EIO08031879806',
	sUserName:= 'ff706992-502b-43c6-8bfd-4102c11712b1', 
	sUserPassword:= 'c02d99ff-a830-4cb7-a7e9-b968a4039aae', 
	eSavePositionCertificate:= eSavePositionOnPLC.ePostionHardDisk, 
	bConnected=> , 
	bError=> , 
	hrErrorCode=> , 
	eConnectionState=> , 
	eErrorMessage_Out=> );

END_PROGRAM

// ---- FBs/FB_Enphase_Helper.TcPOU
FUNCTION_BLOCK FB_Enphase_Helper
VAR_INPUT
	bSend			: BOOL;
END_VAR

VAR_IN_OUT
	fbClient		: FB_IotHttpClient;
END_VAR

VAR_OUTPUT
	bBusy			: BOOL;
	bError			: BOOL;
	lrpowerprod			: LREAL;
	lrpowercons			: LREAL;

END_VAR

VAR
	fbRequestEnphase	: FB_IotHttpRequest;
	fbJson				: FB_JsonDomParser;
	nState				: UDINT;
	RisingEdge			: R_TRIG;
	timTimeout			: TON;
	tTimeOut			: TIME := T#30S;
	
	bGetContentResult	: BOOL;
	sContent			: STRING(2048);
	
	bGetJsonResult		: BOOL;
	jsonDoc				: SJsonValue;
	jsonVal				: SJsonValue;
	
	nReqCount			: UDINT;	
	nResCount			: UDINT;
	nValidResCount		: UDINT;
	nErrCount			: UDINT;
END_VAR

//Timer for Timeout
timTimeout(IN:= nState = 1 AND bBusy, PT:= tTimeOut, Q=> , ET=> );
	IF timTimeout.Q THEN 
		nState := 0;
		bBusy := FALSE;
	END_IF


RisingEdge(CLK:= bSend );


CASE nState OF
0:	
	IF RisingEdge.Q THEN 
		IF
			fbRequestEnphase.SendRequest(sUri:='/production.json', fbClient:=fbClient, eRequestType:=ETcIotHttpRequestType.HTTP_Get, 0, 0, 0) THEN				
				nState:= 1;
				nReqCount:= nReqCount+1;
				bBusy:= TRUE;
				bError:= FALSE;
		END_IF					
	END_IF
	
	
1:
	IF NOT fbRequestEnphase.bBusy THEN
		bError:= TRUE;
		
		IF NOT fbRequestEnphase.bError THEN				 
			bGetContentResult:= fbRequestEnphase.GetContent(pContent:= ADR(sContent), nContentSize:= SIZEOF(sContent), bSetNullTermination:= TRUE);
			IF fbRequestEnphase.nStatusCode >= 200 AND fbRequestEnphase.nStatusCode < 300 THEN
				bGetJsonResult:= FALSE;
				jsonDoc:= fbRequestEnphase.GetJsonDomContent(fbJson);
				IF jsonDoc <> 0 THEN
					bGetJsonResult:= TRUE;
					IF fbJson.HasMember(jsonDoc, 'production')  THEN
						jsonVal:= fbJson.FindMember(jsonDoc, 'production');
						jsonVal:= fbJson.GetArrayValueByIdx(jsonVal, 1);
                        IF fbJson.HasMember(jsonVal, 'wNow') THEN
                            jsonVal:= fbJson.FindMember(jsonVal, 'wNow');
                            nValidResCount:= nValidResCount+1;
                            IF fbJson.IsDouble(jsonVal) THEN
                                lrpowerprod:= fbJson.GetDouble(jsonVal);
                            END_IF
						bError:= FALSE;
						END_IF
					END_IF
					IF fbJson.HasMember(jsonDoc, 'consumption')  THEN
						jsonVal:= fbJson.FindMember(jsonDoc, 'consumption');
						jsonVal:= fbJson.GetArrayValueByIdx(jsonVal, 1);
                        IF fbJson.HasMember(jsonVal, 'wNow') THEN
                            jsonVal:= fbJson.FindMember(jsonVal, 'wNow');
                            nValidResCount:= nValidResCount+1;
                            IF fbJson.IsDouble(jsonVal) THEN
                                lrpowercons:= fbJson.GetDouble(jsonVal);
                            END_IF
						bError:= FALSE;
						END_IF
					END_IF						
				nResCount:= nResCount+1;			
				END_IF
			END_IF
		END_IF
		
	nState:= 0;
	bBusy:= FALSE;
		IF bError THEN
			nErrCount:= nErrCount+1;
		END_IF
	END_IF
	
END_CASE

END_FUNCTION_BLOCK

// ---- FBs/FB_ModBus_2Registers.TcPOU
FUNCTION_BLOCK FB_ModBus_2Registers
VAR_INPUT PERSISTENT
	m_Enable					: BOOL;						//Enable the Fuctionblock and his logic
	str_IPAdress				: STRING(15);				//IP Adress of the meter
	w_Adress					: WORD;						//modbus adress
	int_Divider					: INT;						//Devider of the received data
END_VAR
VAR_OUTPUT
	m_PollSuccessful			: BOOL;						//Poll succesfull		
	r_ReceivedValue				: REAL;						//Received Value
	udint_Error_ID				: UDINT;					// ERR ID FB_MBReadRegs
END_VAR
VAR
	{attribute 'hide'}
	timer_Delay					: TON;						//Timer for Delay between Requests
	{attribute 'hide'}
	timer_DelayStart			: TON;						//Timer to start the state machine with Delay after enabling or after the system ist restartet
	{attribute 'hide'}
	timer_TimeOut				: TON;						//Timer for Timeout MB Read
	{attribute 'hide'}
	iStateModbusRead			: INT;						//State machine for read out Data over Modbus RTU
	{attribute 'hide'}
	fbMBRead_FC3				: FB_MBReadRegs ;		//Modbus Read Function (FC3)
	{attribute 'hide'}
	ftrig_PEnable				: f_trig;					//Internal positive Edge
	{attribute 'hide'}
	iStateModbusError			: INT;						//State machine for error out Data over Modbus TCP/IP	
	{attribute 'hide'}
	FPError_FC_3				: R_TRIG;					//Internal positive Edge
	{attribute 'hide'}
	arrBuffer_FC3				: ARRAY[1..2] OF WORD;		//Buffer with Data from FC3
	{attribute 'hide'}
	timer_Connection_ok			: TON;
	int_Data_Received			: INT;
	{attribute 'hide'}
	m_MBTCPError				: BOOL;
	{attribute 'hide'}
	int_Data_Received_old		: INT;
	{attribute 'hide'}
	timer_Connection_ok_TOF	: TOF;
	{attribute 'hide'}
	fbConvertWordToDword		: FB_CV_WORD_TO_DWORD;			//Convert Word to Dword
	{attribute 'hide'}
	usintSign					: USINT;						// converstion dword to real	
	{attribute 'hide'}
	intExponent					: INT;							// converstion dword to real
	{attribute 'hide'}
	realMantisse				: REAL;							// converstion dword to real
	{attribute 'hide'}
	m_Poll_ok: BOOL;
	{attribute 'hide'}
	timer_Wait: Ton;
	int_TimeoutError: INT;
	int_FC3Error: INT;
END_VAR

(*--------------------------------------------------------------------------------------------Limits-------------------------------------------------------------------------------------*)

w_Adress := LIMIT(0,w_Adress,32767);
int_Divider := LIMIT(1,int_Divider,32767);
	
(*--------------------------------------------------------------------------------------------State Machine Read--------------------------------------------------------------------------------------*)

//Timer for Delay
timer_Delay(IN:= , PT:= T#50MS, Q=> , ET=> );

//Timer for Timeout in Statemachine
IF (iStateModbusRead > 0 AND iStateModbusRead < 3) THEN
	timer_Timeout.IN := TRUE;
ELSE	
	timer_Timeout.IN := FALSE;
END_IF 

//Timeout Timer is dissabled when the Init Step is aktiv or the function is not enabled
IF iStateModbusRead = 0 OR NOT m_Enable THEN 
	timer_Timeout.IN := FALSE; 
END_IF
timer_Timeout(IN:= , PT:= T#1S, Q=> , ET=> );

//Enable with Delay that not all sockets have to be created at the same time
timer_DelayStart(IN:= m_Enable, PT:= T#1S, Q=> , ET=> );
ftrig_PEnable(CLK:= timer_DelayStart.Q, Q=> );

IF ftrig_PEnable.Q AND iStateModbusRead = 0 THEN 
	iStateModbusRead := 1; 
END_IF		
		
//Not Enabled
IF NOT m_Enable THEN 
	iStateModbusRead := 0; 
	iStateModbusError := 0; 
END_IF		
		
CASE iStateModbusRead OF

	0://Init Step 
		timer_Delay.IN := FALSE;
		fbMBRead_FC3.bExecute := FALSE;
		m_Poll_ok:=FALSE;
		int_Data_Received:=0;
	
		iStateModbusRead := 1;
	
	1://read the required registers
		//Start Read
		fbMBRead_FC3.nQuantity := 2;
		fbMBRead_FC3.nMBAddr := w_Adress;
		fbMBRead_FC3.bExecute := TRUE;
		fbMBRead_FC3.nUnitID := 1;
		IF fbMBRead_FC3.bBusy THEN 
			timer_Delay.IN := TRUE; 
		END_IF
		
		//Wait for Delay, copy Data and then next step
		IF NOT fbMBRead_FC3.bBusy AND NOT fbMBRead_FC3.bError AND timer_Delay.Q THEN
			m_Poll_ok:=TRUE;
			int_Data_Received:=int_Data_Received+1;
			m_MBTCPError := FALSE; 
			// convert received data
			
			// dword conversion not tested. Phoenix device sends data in 4 registers
			//		IF m_ConversionToFloat32 = FALSE THEN
			//			fbConvertWordToDword(wInputValue_1:= arrBuffer_FC3[1], wInputValue_2:= arrBuffer_FC3[2], eByteOrderForConvert:= eByteOrder.eLittleEndian, dwOutputValue=> );
			//			r_ReceivedValue := (DWORD_TO_REAL(fbConvertWordToDword.dwOutputValue))/int_Divider;
			//		ELSE
			fbConvertWordToDword(wInputValue_1:= arrBuffer_FC3[1], wInputValue_2:= arrBuffer_FC3[2], eByteOrderForConvert:= eByteOrder.eLittleEndian , dwOutputValue=> );
			(* Sign *)
			usintSign:=BOOL_TO_USINT(fbConvertWordToDword.dwOutputValue.31);
			(* Exponent *)
			intExponent:=DWORD_TO_INT(SHR(fbConvertWordToDword.dwOutputValue,23) AND 16#FF);
			(* Mantisse *)
			realMantisse:=DWORD_TO_REAL(fbConvertWordToDword.dwOutputValue AND 16#7FFFFF);
			(* Result *)
			r_ReceivedValue := LREAL_TO_REAL((EXPT((-1),usintSign) * (1+realMantisse/8388608) * EXPT(2,intExponent-127))/int_Divider);
			//Go to Next Step
			fbMBRead_FC3.bExecute := FALSE;
			timer_Delay.IN := FALSE;		
			iStateModbusRead := 3;
		END_IF	

		//Error or Timeout
		IF FPError_FC_3.Q THEN 
			iStateModbusError := 300;
			int_FC3Error := int_FC3Error+1;
		ELSIF timer_Timeout.Q THEN   	
			iStateModbusError := 300;
			int_TimeoutError := int_TimeoutError+1;
		END_IF
		
	
	3://Wait and go to step 1
		//1 because 0 is the Init Step for Read
		timer_Wait.IN := TRUE;
		
		IF timer_Wait.Q = TRUE THEN
			iStateModbusRead := 1;
			timer_Wait.IN :=FALSE;
		END_IF

			
		
		//Error on Master, changes on Inputs or Timeout
		IF timer_Timeout.Q THEN 
			iStateModbusError := 300; 
		END_IF
	
END_CASE

(* wait timer*)

timer_Wait(PT:=T#3S);


(*------------------------------------------------------------------Error and Warning----------------------------------------------------------------------------*)	
 
timer_Connection_ok			(In:=int_Data_Received<>int_Data_Received_old,PT:=T#10S);
timer_Connection_ok_TOF		(In:=NOT(int_Data_Received<>int_Data_Received_old) AND int_Data_Received>3 ,PT:=T#20S);
int_Data_Received_old:=int_Data_Received;
m_PollSuccessful:=NOT timer_Connection_ok.Q AND timer_Connection_ok_TOF.Q ;

(*------------------------------------------------------------------------------------------Modbus TCP Functions---------------------------------------------------------------------------------------------*)

fbMBRead_FC3(	sIPAddr:= str_IPAdress, 
				nTCPPort:= 502,
				cbLength:= SIZEOF(arrBuffer_FC3), 
				pDestAddr:= ADR(arrBuffer_FC3), 
				tTimeout:= T#10S,
				nErrId => udint_Error_ID);

FPError_FC_3(CLK:= fbMBRead_FC3.  bError, Q=> );		

(*------------------------------------------------------------------------------------------State Machine Error---------------------------------------------------------------------------------------------*)	

CASE iStateModbusError OF
	
	300://Error
		timer_Wait.IN :=TRUE;
		timer_Delay.IN := FALSE;
		fbMBRead_FC3.bExecute := FALSE;
		m_MBTCPError := TRUE; 		
		m_Poll_ok:=FALSE;
		int_Data_Received:=0;
				//Restart from new with the Read out part after an Error
		IF timer_Wait.Q = TRUE THEN
			iStateModbusRead := 0;	
			iStateModbusError := 0;
			timer_Wait.IN :=FALSE;
		END_IF		
							
END_CASE

END_FUNCTION_BLOCK

// ---- POUs/prgBattery.TcPOU
PROGRAM prgBattery
VAR
	fbBatt						: FB_SunSpec_PV_Inverter_T;
	fbBattCounter				: FB_EnergyCounter;
	lrPowerBatt					: LREAL;						//{#lynus.ag#()}
	dwSOCBattery				: DWORD;						//{#lynus.ag#()}
	byErrorWarningBatt			: BYTE;							//{#lynus.ag#()}
END_VAR
VAR PERSISTENT
	lrCounterBatt				: LREAL;						//{#lynus.ag#()}
END_VAR

// To-Do:
// adopt FB Declaration, change to correct FB
// adopt FB Definition, change to correct in/out Vars
// correct lrPowerBatt definition
// correct lrCounterBatt definition
// correct byErrorWarningBatt definition

fbBatt(
	bEnable:= TRUE, 
	sIPAdress:= '192.168.1.25', 
	byUnitID_Inverter:= 1, 
	stDataSunSpec=> , 
	stDataEMPower_PV=> , 
	stDataEMCounter_PV=> , 
	diNrOfEM_OUT_PV=> );

lrPowerBatt := fbBatt.stDataEMPower_PV.lrPowerTotal;
byErrorWarningBatt := fbBatt.stDataEMPower_PV.byErrorWarning;

fbBattCounter(
	byActiveTariff:= 1, 
	lrPowerInput:= lrPowerBatt, 
	lrTotalCounterEnergy_Consumption=> , 
	lrTotalCounterEnergy_Production=> , 
	lrCounterEnergyT1_Consumption=> , 
	lrCounterEnergyT2_Consumption=> , 
	lrCounterEnergyT1_Production=> , 
	lrCounterEnergyT2_Production=> );
	
IF fbBattCounter.lrTotalCounterEnergy_Consumption > lrCounterBatt THEN  	
	lrCounterBatt := fbBattCounter.lrTotalCounterEnergy_Consumption;
END_IF

END_PROGRAM

// ---- POUs/prgPV.TcPOU
PROGRAM prgPV
VAR
	fbPV						: FB_SunSpec_PV_Inverter_T;
	lrPowerPV					: LREAL;						//{#lynus.ag#()}
	byErrorWarningPV			: BYTE;							//{#lynus.ag#()}
END_VAR
VAR PERSISTENT
	lrCounterPV					: LREAL;						//{#lynus.ag#()}
END_VAR

// To-Do:
// adopt FB Declaration, change to correct FB
// adopt FB Definition, change to correct in/out Vars
// correct lrPowerPV definition
// correct lrCounterPV definition
// correct byErrorWarningPV definition

fbPV(
	bEnable:= TRUE, 
	sIPAdress:= '192.168.1.35', 
	byUnitID_Inverter:= 1, 
	stDataSunSpec=> , 
	stDataEMPower_PV=> , 
	stDataEMCounter_PV=> , 
	diNrOfEM_OUT_PV=> );

lrPowerPV := fbPV.stDataEMPower_PV.lrPowerTotal;
byErrorWarningPV := fbPV.stDataEMPower_PV.byErrorWarning;
	
IF fbPV.stDataEMCounter_PV.lrCounterEnergyT1_Production > lrCounterPV THEN  	
	lrCounterPV := fbPV.stDataEMCounter_PV.lrCounterEnergyT1_Production;
END_IF

END_PROGRAM
